(* CoDeSys 2.3 export: MNG_APPLICATION_OUTPUTS_32BIT.EXP *)

(* Data type *)
(*                                                                            *)

TYPE MNG_APPLICATION_OUTPUTS_32BIT :
STRUCT
    NumSignals                    : INT     := 2         ;
    Source01_IN_ISSHOW            : UINT    := 0; (* ics://physics/CGK/InitializePallet/Source?IN_ISSHOW *)
    Source01_IN_LOCATION          : UINT    := 0; (* s://physics/CGK/InitializePallet/Source?IN_LOCATION *)
END_STRUCT
END_TYPE
